PROGRAM P_FeedForward_1
VAR
	
	fbFF : FB_FeedForward;
	
END_VAR

END_PROGRAM

(* stored: Version 1.1.0.1
   POU P_FeedForward_1: Id {06a25b85-bf54-4ee1-9b39-ca8728e6b622}, SpecialFunc None *)
